// TIA Portal V16 export
// export: Created 2021-08-10T09:04:59.8841663Z, ExportSetting WithDefaults, WithReadOnly, DisplayName Totally Integrated Automation Portal, DisplayVersion V16, DisplayName TIA Portal Version Control Interface, DisplayVersion V16, DisplayName TIA Portal Openness, DisplayVersion V16, DisplayName TIA Portal Teamcenter Gateway, DisplayVersion V16, DisplayName SINAMICS Startdrive Advanced, DisplayVersion V16, DisplayName SINAMICS Startdrive G130, G150, S120, S150, SINAMICS MV, S210, DisplayVersion V16, DisplayName SINAMICS Startdrive G110M, G120, G120C, G120D, G120P, DisplayVersion V16, DisplayName STEP 7 Professional, DisplayVersion V16, DisplayName STEP 7 Safety, DisplayVersion V16, DisplayName WinCC Unified SCADA Engineering System, DisplayVersion V16
DATA_BLOCK "Valve Liquid 1_DB"   // DB8
{ S7_Optimized_Access := 'TRUE' }
VERSION : 0.1
// stored: AutoNumber true, CodeModifiedDate 2020-02-26T12:49:41.2445202Z, CompileDate 2021-07-03T08:38:43.2873738Z, CreationDate 2020-02-26T12:48:17.7591506Z, DBAccessibleFromOPCUA true, DownloadWithoutReinit false, InstanceOfName Valve Liquid 1, InstanceOfNumber 2, InstanceOfType FB, InterfaceModifiedDate 2020-02-26T12:49:32.479094Z, IsConsistent true, IsKnowHowProtected false, IsRetainMemResEnabled false, MemoryReserve 100, ModifiedDate 2020-02-26T12:49:41.2445202Z, ParameterModified 2020-02-26T07:16:31.1886327Z, StructureModified 2020-02-26T12:49:32.479094Z, UDAEnableTagReadback false
"Valve Liquid 1"
   // VAR
   //    VlvLiq1 : "fbValve_Solenoid";
   // END_VAR
BEGIN
END_DATA_BLOCK
